KUKA KRL program: Safety_Position.src, Safety_Position.dat

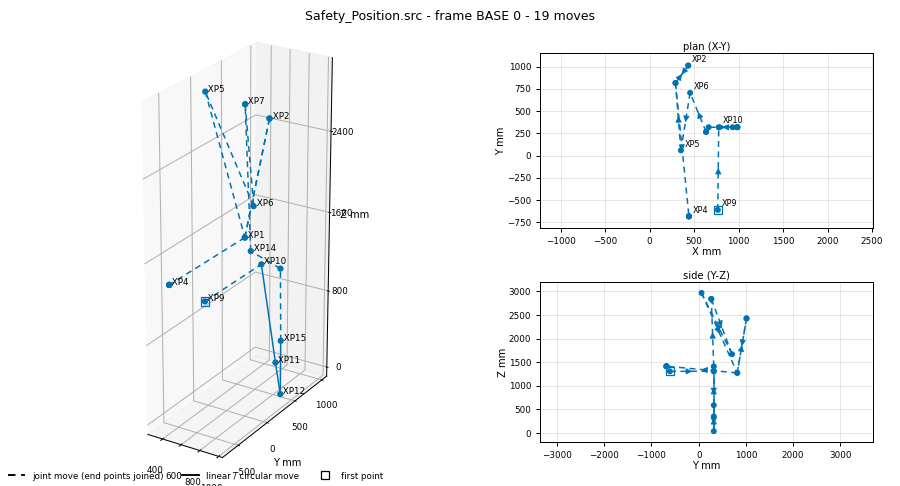
[picture p0: tool path of Safety_Position.src in frame BASE 0, 19 of 19 moves have a stored position in this frame; points joined in program order, loops and branches not executed]
--- Safety_Position.src ---
&ACCESS RVP1
&REL 76
&COMMENT Safety Position
&PARAM DISKPATH = KRC:\R1\Program\Safety Programs
DEF SAFETY_POSITION(DIRECTION :IN,AREA_NR :IN,TYPE_NR :IN )
;FOLD INI
  INT DIRECTION
  INT AREA_NR
  INT TYPE_NR
  decl KrlMsg_T msg
  decl KrlMsgPar_T par[3]
  decl KrlMsgOpt_T opt
  INT nHandle

  IF (DIRECTION>2) OR (DIRECTION<1) THEN
    REPEAT
      msg = {modul[] "Safety Position", nr 1, msg_txt[] "Direction Number Not Valid"}

			opt = {vl_stop true, clear_p_reset true, clear_p_SAW false, log_to_DB false}

			nHandle = Set_KrlMsg(#notify, msg, par[], opt)
      HALT
    UNTIL (DIRECTION<3) AND (DIRECTION>0)
  ENDIF
  IF (AREA_NR>8) OR (AREA_NR<1) THEN
    REPEAT
      msg = {modul[] "Safety Position", nr 2, msg_txt[] "Area Number Not Valid"}

			opt = {vl_stop true, clear_p_reset true, clear_p_SAW false, log_to_DB false}

			nHandle = Set_KrlMsg(#notify, msg, par[], opt)
      HALT
    UNTIL (AREA_NR<9) AND (AREA_NR>0)
  ENDIF
  IF (TYPE_NR>8) OR (TYPE_NR<1) THEN
    REPEAT
  	  msg = {modul[] "Safety Position", nr 1, msg_txt[] "Type Number Not Valid"}

			opt = {vl_stop true, clear_p_reset true, clear_p_SAW false, log_to_DB false}

			nHandle = Set_KrlMsg(#notify, msg, par[], opt)
      HALT
    UNTIL (TYPE_NR<9) AND (TYPE_NR>0)
  ENDIF
  ;ENDFOLD
;===================================================
; MODEL     :CX482
; IE GROUP  :PHEV
; STATION   :110
; ROBOT     :110R1
; FUNCTION  : Safety Position
;================================================

SWITCH AREA_NR

CASE 1  ;AREA 1

  SWITCH TYPE_NR

  CASE 1  ;Area 1 - Safety Position 1
    SWITCH DIRECTION
    CASE 1
    ;Teach here positions from wait area to safety position
    ;check robot movement for collision with other robots
;FOLD PTP P9 CONT Vel=100 % PDAT17 Tool[8]:Gripper_array Base[0];%{PE}%R 8.3.48,%MKUKATPBASIS,%CMOVE,%VPTP,%P 1:PTP, 2:P9, 3:C_DIS, 5:100, 7:PDAT17
$BWDSTART=FALSE
PDAT_ACT=PPDAT17
FDAT_ACT=FP9
BAS(#PTP_PARAMS,100)
PTP XP9 C_DIS
;ENDFOLD
;FOLD PTP P10 CONT Vel=100 % PDAT18 Tool[8]:Gripper_array Base[0];%{PE}%R 8.3.48,%MKUKATPBASIS,%CMOVE,%VPTP,%P 1:PTP, 2:P10, 3:C_DIS, 5:100, 7:PDAT18
$BWDSTART=FALSE
PDAT_ACT=PPDAT18
FDAT_ACT=FP10
BAS(#PTP_PARAMS,100)
PTP XP10 C_DIS
;ENDFOLD
;FOLD LIN P11 CONT Vel=2 m/s CPDAT1 Tool[8]:Gripper_array Base[0];%{PE}%R 8.3.48,%MKUKATPBASIS,%CMOVE,%VLIN,%P 1:LIN, 2:P11, 3:C_DIS C_DIS, 5:2, 7:CPDAT1
$BWDSTART=FALSE
LDAT_ACT=LCPDAT1
FDAT_ACT=FP11
BAS(#CP_PARAMS,2)
LIN XP11 C_DIS C_DIS
;ENDFOLD
;FOLD LIN P12 Vel=2 m/s CPDAT2 Tool[8]:Gripper_array Base[0];%{PE}%R 8.3.48,%MKUKATPBASIS,%CMOVE,%VLIN,%P 1:LIN, 2:P12, 3:, 5:2, 7:CPDAT2
$BWDSTART=FALSE
LDAT_ACT=LCPDAT2
FDAT_ACT=FP12
BAS(#CP_PARAMS,2)
LIN XP12
;ENDFOLD

;abrir gara
cil_bat_reposo()


;FOLD LIN P15 CONT Vel=2 m/s CPDAT3 Tool[8]:Gripper_array Base[0];%{PE}%R 8.3.48,%MKUKATPBASIS,%CMOVE,%VLIN,%P 1:LIN, 2:P15, 3:C_DIS C_DIS, 5:2, 7:CPDAT3
$BWDSTART=FALSE
LDAT_ACT=LCPDAT3
FDAT_ACT=FP15
BAS(#CP_PARAMS,2)
LIN XP15 C_DIS C_DIS
;ENDFOLD
;FOLD PTP P13 CONT Vel=100 % PDAT19 Tool[8]:Gripper_array Base[0];%{PE}%R 8.3.48,%MKUKATPBASIS,%CMOVE,%VPTP,%P 1:PTP, 2:P13, 3:C_DIS, 5:100, 7:PDAT19
$BWDSTART=FALSE
PDAT_ACT=PPDAT19
FDAT_ACT=FP13
BAS(#PTP_PARAMS,100)
PTP XP13 C_DIS
;ENDFOLD
;FOLD PTP P14 CONT Vel=100 % PDAT20 Tool[8]:Gripper_array Base[0];%{PE}%R 8.3.48,%MKUKATPBASIS,%CMOVE,%VPTP,%P 1:PTP, 2:P14, 3:C_DIS, 5:100, 7:PDAT20
$BWDSTART=FALSE
PDAT_ACT=PPDAT20
FDAT_ACT=FP14
BAS(#PTP_PARAMS,100)
PTP XP14 C_DIS
;ENDFOLD

;FOLD PTP P7 Vel=100 % PDAT15 Tool[8]:Gripper_array Base[0];%{PE}%R 8.3.48,%MKUKATPBASIS,%CMOVE,%VPTP,%P 1:PTP, 2:P7, 3:, 5:100, 7:PDAT15
$BWDSTART=FALSE
PDAT_ACT=PPDAT15
FDAT_ACT=FP7
BAS(#PTP_PARAMS,100)
PTP XP7
;ENDFOLD
    CASE 2
    ;Teach here positions from safety position to wait area
;FOLD PTP P8 CONT Vel=100 % PDAT16 Tool[8]:Gripper_array Base[0];%{PE}%R 8.3.48,%MKUKATPBASIS,%CMOVE,%VPTP,%P 1:PTP, 2:P8, 3:C_DIS, 5:100, 7:PDAT16
$BWDSTART=FALSE
PDAT_ACT=PPDAT16
FDAT_ACT=FP8
BAS(#PTP_PARAMS,100)
PTP XP8 C_DIS
;ENDFOLD
    ;check robot movement for collision with other robots
    ENDSWITCH

  CASE 2  ;Area 1 - Safety Position 2

    SWITCH DIRECTION
    CASE 1
;FOLD PTP P6 CONT Vel=100 % PDAT14 Tool[1] Base[0];%{PE}%R 8.3.48,%MKUKATPBASIS,%CMOVE,%VPTP,%P 1:PTP, 2:P6, 3:C_DIS, 5:100, 7:PDAT14
$BWDSTART=FALSE
PDAT_ACT=PPDAT14
FDAT_ACT=FP6
BAS(#PTP_PARAMS,100)
PTP XP6 C_DIS
;ENDFOLD
;FOLD PTP P5 Vel=100 % PDAT13 Tool[1] Base[0];%{PE}%R 8.3.48,%MKUKATPBASIS,%CMOVE,%VPTP,%P 1:PTP, 2:P5, 3:, 5:100, 7:PDAT13
$BWDSTART=FALSE
PDAT_ACT=PPDAT13
FDAT_ACT=FP5
BAS(#PTP_PARAMS,100)
PTP XP5
;ENDFOLD
    ;Teach here positions from waiting area to safety position
    ;check robot movement for collision with other robots
;FOLD PTP P1 Vel=100 % PDAT5 Tool[8]:Gripper_array Base[0];%{PE}%R 8.3.48,%MKUKATPBASIS,%CMOVE,%VPTP,%P 1:PTP, 2:P1, 3:, 5:100, 7:PDAT5
$BWDSTART=FALSE
PDAT_ACT=PPDAT5
FDAT_ACT=FP1
BAS(#PTP_PARAMS,100)
PTP XP1
;ENDFOLD
;FOLD PTP P2 Vel=100 % PDAT6 Tool[8]:Gripper_array Base[0];%{PE}%R 8.3.48,%MKUKATPBASIS,%CMOVE,%VPTP,%P 1:PTP, 2:P2, 3:, 5:100, 7:PDAT6
$BWDSTART=FALSE
PDAT_ACT=PPDAT6
FDAT_ACT=FP2
BAS(#PTP_PARAMS,100)
PTP XP2
;ENDFOLD
    CASE 2
    ;Teach here positions from safety position to waiting area
    ;check robot movement for collision with other robots
;FOLD PTP P2 Vel=100 % PDAT7 Tool[8]:Gripper_array Base[0];%{PE}%R 8.3.48,%MKUKATPBASIS,%CMOVE,%VPTP,%P 1:PTP, 2:P2, 3:, 5:100, 7:PDAT7
$BWDSTART=FALSE
PDAT_ACT=PPDAT7
FDAT_ACT=FP2
BAS(#PTP_PARAMS,100)
PTP XP2
;ENDFOLD
;FOLD PTP P1 Vel=100 % PDAT8 Tool[8]:Gripper_array Base[0];%{PE}%R 8.3.48,%MKUKATPBASIS,%CMOVE,%VPTP,%P 1:PTP, 2:P1, 3:, 5:100, 7:PDAT8
$BWDSTART=FALSE
PDAT_ACT=PPDAT8
FDAT_ACT=FP1
BAS(#PTP_PARAMS,100)
PTP XP1
;ENDFOLD
    ENDSWITCH

  CASE 3  ;Area 1 - Safety Position 3

    SWITCH DIRECTION
    CASE 1
    ;Teach here positions from waiting area to safety position
    ;check robot movement for collision with other robots
;FOLD PTP P4 Vel=100 % PDAT10 Tool[8]:Gripper_array Base[0];%{PE}%R 8.3.48,%MKUKATPBASIS,%CMOVE,%VPTP,%P 1:PTP, 2:P4, 3:, 5:100, 7:PDAT10
$BWDSTART=FALSE
PDAT_ACT=PPDAT10
FDAT_ACT=FP4
BAS(#PTP_PARAMS,100)
PTP XP4
;ENDFOLD
;FOLD PTP P3 Vel=100 % PDAT9 Tool[8]:Gripper_array Base[0];%{PE}%R 8.3.48,%MKUKATPBASIS,%CMOVE,%VPTP,%P 1:PTP, 2:P3, 3:, 5:100, 7:PDAT9
$BWDSTART=FALSE
PDAT_ACT=PPDAT9
FDAT_ACT=FP3
BAS(#PTP_PARAMS,100)
PTP XP3
;ENDFOLD
    CASE 2
    ;Teach here positions from safety position to waiting area
    ;check robot movement for collision with other robots
;FOLD PTP P3 Vel=100 % PDAT11 Tool[8]:Gripper_array Base[0];%{PE}%R 8.3.48,%MKUKATPBASIS,%CMOVE,%VPTP,%P 1:PTP, 2:P3, 3:, 5:100, 7:PDAT11
$BWDSTART=FALSE
PDAT_ACT=PPDAT11
FDAT_ACT=FP3
BAS(#PTP_PARAMS,100)
PTP XP3
;ENDFOLD
;FOLD PTP P4 Vel=100 % PDAT12 Tool[8]:Gripper_array Base[0];%{PE}%R 8.3.48,%MKUKATPBASIS,%CMOVE,%VPTP,%P 1:PTP, 2:P4, 3:, 5:100, 7:PDAT12
$BWDSTART=FALSE
PDAT_ACT=PPDAT12
FDAT_ACT=FP4
BAS(#PTP_PARAMS,100)
PTP XP4
;ENDFOLD
    ENDSWITCH

  CASE 4  ;Area 1 - Safety Position 4

    SWITCH DIRECTION
    CASE 1 ; From Area Request Position To Safety Position
    ;Teach here positions from waiting area to safety position
    ;check robot movement for collision with other robots
    CASE 2 ; From Safety Position To Area Request Position
    ;Teach here positions from safety position to waiting area
    ;check robot movement for collision with other robots
    ENDSWITCH

  CASE 5  ;Area 1 - Safety Position 5

    SWITCH DIRECTION
    CASE 1
    ;Teach here positions from waiting area to safety position
    ;check robot movement for collision with other robots
    CASE 2
    ;Teach here positions from safety position to waiting area
    ;check robot movement for collision with other robots
    ENDSWITCH

  CASE 6  ;Area 1 - Safety Position 6

    SWITCH DIRECTION
    CASE 1
    ;Teach here positions from waiting area to safety position
    ;check robot movement for collision with other robots
    CASE 2
    ;Teach here positions from safety position to waiting area
    ;check robot movement for collision with other robots
    ENDSWITCH

  CASE 7  ;Area 1 - Safety Position 7

    SWITCH DIRECTION
    CASE 1
    ;Teach here positions from waiting area to safety position
    ;check robot movement for collision with other robots
    CASE 2
    ;Teach here positions from safety position to waiting area
    ;check robot movement for collision with other robots
    ENDSWITCH

  CASE 8  ;Area 1 - Safety Position 8

    SWITCH DIRECTION
    CASE 1
    ;Teach here positions from wait area to safety position
    ;check robot movement for collision with other robots
    CASE 2
    ;Teach here positions from safety position to wait area
    ;check robot movement for collision with other robots
    ENDSWITCH

  ENDSWITCH

;====================================================================

CASE 2  ;AREA 2

  SWITCH TYPE_NR
  CASE 1  ;Area 2 - Safety Position 1

    SWITCH DIRECTION
    CASE 1
    ;Teach here pos from waiting area to safety position
    ;check robot movement for collision with other robots
    CASE 2
    ;Teach here positions from safety pos to waiting area
    ;check robot movement for collision with other robots
    ENDSWITCH

  CASE 2  ;Area 2 - Safety Position 2

    SWITCH DIRECTION
    CASE 1
    ;Teach here positions from waiting area to safety position
    ;check robot movement for collision with other robots
    CASE 2
    ;Teach here positions from safety position to waiting area
    ;check robot movement for collision with other robots
    ENDSWITCH

  CASE 3  ;Area 2 - Safety Position 3

    SWITCH DIRECTION
    CASE 1
    ;Teach here positions from waiting area to safety position
    ;check robot movement for collision with other robots
    CASE 2
    ;Teach here positions from safety position to waiting area
    ;check robot movement for collision with other robots
    ENDSWITCH

  CASE 4  ;Area 2 - Safety Position 4

    SWITCH DIRECTION
	  	CASE 1
    ;Teach here positions from waiting area to safety position
    ;check robot movement for collision with other robots
    CASE 2
    ;Teach here positions from safety position to waiting area
    ;check robot movement for collision with other robots
    ENDSWITCH

  CASE 5  ;Area 2 - Safety Position 5

    SWITCH DIRECTION
    CASE 1
    ;Teach here positions from waiting area to safety position
    ;check robot movement for collision with other robots
    CASE 2
    ;Teach here positions from safety position to waiting area
    ;check robot movement for collision with other robots
    ENDSWITCH

  CASE 6    ;Area 2 - Safety Position 6

    SWITCH DIRECTION
    CASE 1
    ;Teach here positions from waiting area to safety position
    ;check robot movement for collision with other robots
    CASE 2
    ;Teach here positions from safety position to waiting area
    ;check robot movement for collision with other robots
    ENDSWITCH

  CASE 7    ;Area 2 - Safety Position 7

    SWITCH DIRECTION
    CASE 1
    ;Teach here positions from waiting area to safety position
    ;check robot movement for collision with other robots
    CASE 2
    ;Teach here positions from safety position to waiting area
    ;check robot movement for collision with other robots
    ENDSWITCH

  CASE 8  ;Area 2 - Safety Position 8

    SWITCH DIRECTION
    CASE 1
    ;Teach here positions from waiting area to safety position
    ;check robot movement for collision with other robots
    CASE 2
    ;Teach here positions from safety position to waiting area
    ;check robot movement for collision with other robots
    ENDSWITCH

  ENDSWITCH

;====================================================================

CASE 3  ;AREA 3

  SWITCH TYPE_NR
  CASE 1  ;Area 3 - Safety Position 1

    SWITCH DIRECTION
    CASE 1
    ;Teach here positions from waiting area to safety position
    ;check robot movement for collision with other robots
    CASE 2
    ;Teach here positions from safety position to waiting area
    ;check robot movement for collision with other robots
    ENDSWITCH

  CASE 2  ;Area 3 - Safety Position 2

    SWITCH DIRECTION
    CASE 1
    ;Teach here positions from waiting area to safety position
    ;check robot movement for collision with other robots
    CASE 2
    ;Teach here positions from safety position to waiting area
    ;check robot movement for collision with other robots
    ENDSWITCH

  CASE 3  ;Area 3 - Safety Position 3

    SWITCH DIRECTION
    CASE 1
    ;Teach here positions from waiting area to safety position
    ;check robot movement for collision with other robots
    CASE 2
    ;Teach here positions from safety position to waiting area
    ;check robot movement for collision with other robots
      ENDSWITCH

  CASE 4  ;Area 3 - Safety Position 4

    SWITCH DIRECTION
    CASE 1
    ;Teach here positions from waiting area to safety position
    ;check robot movement for collision with other robots
    CASE 2
    ;Teach here positions from safety position to waiting area
    ;check robot movement for collision with other robots
    ENDSWITCH

  CASE 5  ;Area 3 - Safety Position 5

    SWITCH DIRECTION
    CASE 1
    ;Teach here positions from waiting area to safety position
    ;check robot movement for collision with other robots
    CASE 2
    ;Teach here positions from safety position to waiting area
    ;check robot movement for collision with other robots
    ENDSWITCH

  CASE 6  ;Area 3 - Safety Position 6

    SWITCH DIRECTION
    CASE 1
    ;Teach here positions from waiting area to safety position
    ;check robot movement for collision with other robots
    CASE 2
    ;Teach here positions from safety position to waiting area
    ;check robot movement for collision with other robots
    ENDSWITCH

  CASE 7  ;Area 3 - Safety Position 7

    SWITCH DIRECTION
    CASE 1
    ;Teach here positions from waiting area to safety position
    ;check robot movement for collision with other robots
    CASE 2
    ;Teach here positions from safety position to waiting area
    ;check robot movement for collision with other robots
    ENDSWITCH

  CASE 8  ;Area 3 - Safety Position 8
    SWITCH DIRECTION
    CASE 1
    ;Teach here positions from waiting area to safety position
    ;check robot movement for collision with other robots
    CASE 2
    ;Teach here positions from safety position to waiting area
    ;check robot movement for collision with other robots
    ENDSWITCH

  ENDSWITCH

;====================================================================

CASE 4  ;AREA 4

  SWITCH TYPE_NR
  CASE 1  ;Area 4 - Safety Position 1

    SWITCH DIRECTION
    CASE 1
		;Teach here positions from waiting area to safety position
		;check robot movement for collision with other robots
		CASE 2
		;Teach here positions from safety position to waiting area
		;check robot movement for collision with other robots

    ENDSWITCH

  CASE 2  ;Area 4 - Safety Position 2

    SWITCH DIRECTION
    CASE 1
	  ;Teach here positions from waiting area to safety position
	  ;check robot movement for collision with other robots
    CASE 2
	  ;Teach here positions from safety position to waiting area
  	;check robot movement for collision with other robots
    ENDSWITCH

  CASE 3  ;Area 4 - Safety Position 3

    SWITCH DIRECTION
    CASE 1
    ;Teach here positions from waiting area to safety position
    ;check robot movement for collision with other robots
    CASE 2
    ;Teach here positions from safety position to waiting area
    ;check robot movement for collision with other robots
    ENDSWITCH

  CASE 4  ;Area 4 - Safety Position 4

    SWITCH DIRECTION
    CASE 1
    ;Teach here positions from waiting area to safety position
    ;check robot movement for collision with other robots
    CASE 2
    ;Teach here positions from safety position to waiting area
    ;check robot movement for collision with other robots
    ENDSWITCH

  CASE 5  ;Area 4 - Safety Position 5

    SWITCH DIRECTION
    CASE 1
    ;Teach here positions from waiting area to safety position
    ;check robot movement for collision with other robots
    CASE 2
    ;Teach here positions from safety position to waiting area
    ;check robot movement for collision with other robots
    ENDSWITCH

  CASE 6  ;Area 4 - Safety Position 6

    SWITCH DIRECTION
    CASE 1
    ;Teach here positions from waiting area to safety position
    ;check robot movement for collision with other robots
    CASE 2
    ;Teach here positions from safety position to waiting area
    ;check robot movement for collision with other robots
    ENDSWITCH

  CASE 7  ;Area 4 - Safety Position 7

    SWITCH DIRECTION
    CASE 1
    ;Teach here positions from waiting area to safety position
    ;check robot movement for collision with other robots
    CASE 2
    ;Teach here positions from safety position to waiting area
    ;check robot movement for collision with other robots
    ENDSWITCH

  CASE 8  ;Area 4 - Safety Position 8

    SWITCH DIRECTION
    CASE 1
    ;Teach here positions from waiting area to safety position
    ;check robot movement for collision with other robots
    CASE 2
    ;Teach here positions from safety position to waiting area
    ;check robot movement for collision with other robots
    ENDSWITCH

  ENDSWITCH

;====================================================================

CASE 5  ;AREA 5

  SWITCH TYPE_NR
  CASE 1  ;Area 5 - Safety Position 1

    SWITCH DIRECTION
    CASE 1
    ;Teach here positions from waiting area to safety position
    ;check robot movement for collision with other robots
    CASE 2
    ;Teach here positions from safety position to waiting area
    ;check robot movement for collision with other robots
    ENDSWITCH

  CASE 2  ;Area 5 - Safety Position 2

    SWITCH DIRECTION
    CASE 1
    ;Teach here positions from waiting area to safety position
    ;check robot movement for collision with other robots
    CASE 2
    ;Teach here positions from safety position to waiting area
    ;check robot movement for collision with other robots
    ENDSWITCH

  CASE 3  ;Area 5 - Safety Position 3

    SWITCH DIRECTION
    CASE 1
    ;Teach here positions from waiting area to safety position
    ;check robot movement for collision with other robots
    CASE 2
    ;Teach here positions from safety position to waiting area
    ;check robot movement for collision with other robots
    ENDSWITCH

  CASE 4  ;Area 5 - Safety Position 4

    SWITCH DIRECTION
    CASE 1
    ;Teach here positions from waiting area to safety position
    ;check robot movement for collision with other robots
    CASE 2
    ;Teach here positions from safety position to waiting area
    ;check robot movement for collision with other robots
    ENDSWITCH

  CASE 5  ;Area 5 - Safety Position 5

    SWITCH DIRECTION
    CASE 1
    ;Teach here positions from waiting area to safety position
    ;check robot movement for collision with other robots
    CASE 2
    ;Teach here positions from safety position to waiting area
    ;check robot movement for collision with other robots
    ENDSWITCH

  CASE 6  ;Area 5 - Safety Position 6

    SWITCH DIRECTION
    CASE 1
    ;Teach here positions from waiting area to safety position
    ;check robot movement for collision with other robots
    CASE 2
    ;Teach here positions from safety position to waiting area
    ;check robot movement for collision with other robots
    ENDSWITCH

  CASE 7  ;Area 5 - Safety Position 7

    SWITCH DIRECTION
    CASE 1
    ;Teach here positions from waiting area to safety position
    ;check robot movement for collision with other robots
    CASE 2
    ;Teach here positions from safety position to waiting area
    ;check robot movement for collision with other robots
    ENDSWITCH

  CASE 8  ;Area 5 - Safety Position 8

    SWITCH DIRECTION
    CASE 1
    ;Teach here positions from waiting area to safety position
    ;check robot movement for collision with other robots
    CASE 2
    ;Teach here positions from safety position to waiting area
    ;check robot movement for collision with other robots
    ENDSWITCH

  ENDSWITCH

;====================================================================

CASE 6  ;AREA 6

  SWITCH TYPE_NR
  CASE 1  ;Area 6 - Safety Position 1

    SWITCH DIRECTION
    CASE 1
    ;Teach here positions from waiting area to safety position
    ;check robot movement for collision with other robots
    CASE 2
    ;Teach here positions from safety position to waiting area
    ;check robot movement for collision with other robots
    ENDSWITCH

  CASE 2  ;Area 6 - Safety Position 2

    SWITCH DIRECTION
    CASE 1
    ;Teach here positions from waiting area to safety position
    ;check robot movement for collision with other robots
    CASE 2
    ;Teach here positions from safety position to waiting area
    ;check robot movement for collision with other robots
    ENDSWITCH

  CASE 3  ;Area 6 - Safety Position 3

    SWITCH DIRECTION
    CASE 1
    ;Teach here positions from waiting area to safety position
    ;check robot movement for collision with other robots
    CASE 2
    ;Teach here positions from safety position to waiting area
    ;check robot movement for collision with other robots
    ENDSWITCH

  CASE 4  ;Area 6 - Safety Position 4

    SWITCH DIRECTION
    CASE 1
    ;Teach here positions from waiting area to safety position
    ;check robot movement for collision with other robots
    CASE 2
    ;Teach here positions from safety position to waiting area
    ;check robot movement for collision with other robots
    ENDSWITCH

  CASE 5  ;Area 6 - Safety Position 5

    SWITCH DIRECTION
    CASE 1
    ;Teach here positions from waiting area to safety position
    ;check robot movement for collision with other robots
    CASE 2
    ;Teach here positions from safety position to waiting area
    ;check robot movement for collision with other robots
    ENDSWITCH

  CASE 6  ;Area 6 - Safety Position 6

    SWITCH DIRECTION
    CASE 1
    ;Teach here positions from waiting area to safety position
    ;check robot movement for collision with other robots
    CASE 2
    ;Teach here positions from safety position to waiting area
    ;check robot movement for collision with other robots
    ENDSWITCH

  CASE 7  ;Area 6 - Safety Position 7

    SWITCH DIRECTION
    CASE 1
    ;Teach here positions from waiting area to safety position
    ;check robot movement for collision with other robots
    CASE 2
    ;Teach here positions from safety position to waiting area
    ;check robot movement for collision with other robots
    ENDSWITCH

  CASE 8  ;Area 6 - Safety Position 8

    SWITCH DIRECTION
    CASE 1
    ;Teach here positions from waiting area to safety position
    ;check robot movement for collision with other robots
    CASE 2
    ;Teach here positions from safety position to waiting area
    ;check robot movement for collision with other robots
    ENDSWITCH

  ENDSWITCH

;====================================================================

CASE 7  ;AREA 7

  SWITCH TYPE_NR
  CASE 1  ;Area 7 - Safety Position 1

    SWITCH DIRECTION
    CASE 1
    ;Teach here positions from waiting area to safety position
    ;check robot movement for collision with other robots
    CASE 2
    ;Teach here positions from safety position to waiting area
    ;check robot movement for collision with other robots
    ENDSWITCH

  CASE 2  ;Area 7 - Safety Position 2

    SWITCH DIRECTION
    CASE 1
    ;Teach here positions from waiting area to safety position
    ;check robot movement for collision with other robots
    CASE 2
    ;Teach here positions from safety position to waiting area
    ;check robot movement for collision with other robots
    ENDSWITCH

  CASE 3  ;Area 7 - Safety Position 3

    SWITCH DIRECTION
    CASE 1
    ;Teach here positions from waiting area to safety position
    ;check robot movement for collision with other robots
    CASE 2
    ;Teach here positions from safety position to waiting area
    ;check robot movement for collision with other robots
    ENDSWITCH

  CASE 4  ;Area 7 - Safety Position 4

    SWITCH DIRECTION
    CASE 1
    ;Teach here positions from waiting area to safety position
    ;check robot movement for collision with other robots
    CASE 2
    ;Teach here positions from safety position to waiting area
    ;check robot movement for collision with other robots
    ENDSWITCH

  CASE 5  ;Area 7 - Safety Position 5

    SWITCH DIRECTION
    CASE 1
    ;Teach here positions from waiting area to safety position
    ;check robot movement for collision with other robots
    CASE 2
    ;Teach here positions from safety position to waiting area
    ;check robot movement for collision with other robots
    ENDSWITCH

  CASE 6  ;Area 7 - Safety Position 6

    SWITCH DIRECTION
    CASE 1
    ;Teach here positions from waiting area to safety position
    ;check robot movement for collision with other robots
    CASE 2
    ;Teach here positions from safety position to waiting area
    ;check robot movement for collision with other robots
    ENDSWITCH

  CASE 7  ;Area 7 - Safety Position 7

    SWITCH DIRECTION
    CASE 1
    ;Teach here positions from waiting area to safety position
    ;check robot movement for collision with other robots
    CASE 2
    ;Teach here positions from safety position to waiting area
    ;check robot movement for collision with other robots
    ENDSWITCH

  CASE 8  ;Area 7 - Safety Position 8

    SWITCH DIRECTION
    CASE 1
    ;Teach here positions from waiting area to safety position
    ;check robot movement for collision with other robots
    CASE 2
    ;Teach here positions from safety position to waiting area
    ;check robot movement for collision with other robots
    ENDSWITCH

  ENDSWITCH

;====================================================================

CASE 8  ;AREA 8

  SWITCH TYPE_NR
  CASE 1  ;Area 8 - Safety Position 1

    SWITCH DIRECTION
    CASE 1
    ;Teach here positions from waiting area to safety position
    ;check robot movement for collision with other robots
    CASE 2
    ;Teach here positions from safety position to waiting area
    ;check robot movement for collision with other robots
    ENDSWITCH

  CASE 2  ;Area 8 - Safety Position 2

    SWITCH DIRECTION
    CASE 1
    ;Teach here positions from waiting area to safety position
    ;check robot movement for collision with other robots
    CASE 2
    ;Teach here positions from safety position to waiting area
    ;check robot movement for collision with other robots
    ENDSWITCH

  CASE 3  ;Area 8 - Safety Position 3

    SWITCH DIRECTION
    CASE 1
    ;Teach here positions from waiting area to safety position
    ;check robot movement for collision with other robots
    CASE 2
    ;Teach here positions from safety position to waiting area
    ;check robot movement for collision with other robots
    ENDSWITCH

  CASE 4  ;Area 8 - Safety Position 4

    SWITCH DIRECTION
    CASE 1
    ;Teach here positions from waiting area to safety position
    ;check robot movement for collision with other robots
    CASE 2
    ;Teach here positions from safety position to waiting area
    ;check robot movement for collision with other robots
    ENDSWITCH

  CASE 5  ;Area 8 - Safety Position 5

    SWITCH DIRECTION
    CASE 1
    ;Teach here positions from waiting area to safety position
    ;check robot movement for collision with other robots
    CASE 2
    ;Teach here positions from safety position to waiting area
    ;check robot movement for collision with other robots
    ENDSWITCH

  CASE 6  ;Area 8 - Safety Position 6

    SWITCH DIRECTION
    CASE 1
    ;Teach here positions from waiting area to safety position
    ;check robot movement for collision with other robots
    CASE 2
    ;Teach here positions from safety position to waiting area
    ;check robot movement for collision with other robots
    ENDSWITCH

  CASE 7  ;Area 8 - Safety Position 7

    SWITCH DIRECTION
    CASE 1
    ;Teach here positions from waiting area to safety position
    ;check robot movement for collision with other robots
    CASE 2
    ;Teach here positions from safety position to waiting area
    ;check robot movement for collision with other robots
    ENDSWITCH

  CASE 8  ;Area 8 - Safety Position 8

    SWITCH DIRECTION
    CASE 1
    ;Teach here positions from waiting area to safety position
    ;check robot movement for collision with other robots
    CASE 2
    ;Teach here positions from safety position to waiting area
    ;check robot movement for collision with other robots
    ENDSWITCH
  ENDSWITCH
ENDSWITCH
END

--- Safety_Position.dat ---
&ACCESS RVP1
&REL 76
&COMMENT Safety Position
&PARAM DISKPATH = KRC:\R1\Program\Safety Programs
DEFDAT  Safety_Position
;FOLD EXTERNAL DECLARATIONS;%{PE}%V3.2.0,%MKUKATPBASIS,%CEXT,%VCOMMON,%P
;FOLD BAS EXT;%{PE}%V3.2.0,%MKUKATPBASIS,%CEXT,%VEXT,%P
EXT  BAS (BAS_COMMAND  :IN,REAL  :IN )
DECL INT SUCCESS
;ENDFOLD
;FOLD GRIPPERTECH EXT
EXT  H50 (INT  :IN,INT  :IN,INT  :IN,GRP_TYP  :IN )
;ENDFOLD (GRIPPERTECH EXT)
;FOLD SPOTTECH EXT
EXT  USERSPOT (S_COMMAND  :IN,SPOT_TYPE  :IN )
;ENDFOLD (SPOTTECH EXT)
;FOLD USER EXT;%{E}%V3.2.0,%MKUKATPUSER,%CEXT,%VEXT,%P
;Make here your modifications
;ENDFOLD
;ENDFOLD

DECL BASIS_SUGG_T LAST_BASIS={POINT1[] "P15                     ",POINT2[] "P15                     ",CP_PARAMS[] "CPDAT3                  ",PTP_PARAMS[] "PDAT20                  ",CONT[] "C_DIS C_DIS             ",CP_VEL[] "2                       ",PTP_VEL[] "100                     ",SYNC_PARAMS[] "SYNCDAT                 ",SPL_NAME[] "S0                      ",A_PARAMS[] "ADAT0                   "}
DECL E6POS XP1={X 290.951233,Y 816.177124,Z 1275.55042,A -86.9976196,B 22.0779018,C -179.006119,S 6,T 27,E1 0.0,E2 0.0,E3 0.0,E4 0.0,E5 0.0,E6 0.0}
DECL FDAT FP1={TOOL_NO 8,BASE_NO 0,IPO_FRAME #BASE,POINT2[] " ",TQ_STATE FALSE}
DECL PDAT PPDAT1={VEL 100.000,ACC 100.000,APO_DIST 100.000,GEAR_JERK 50.0000,EXAX_IGN 0}
DECL E6POS XP2={X 434.240051,Y 1012.69025,Z 2428.93188,A -59.3382492,B 50.5025139,C -135.088516,S 6,T 27,E1 0.0,E2 0.0,E3 0.0,E4 0.0,E5 0.0,E6 0.0}
DECL FDAT FP2={TOOL_NO 8,BASE_NO 0,IPO_FRAME #BASE,POINT2[] " ",TQ_STATE FALSE}
DECL PDAT PPDAT2={VEL 100.000,ACC 100.000,APO_DIST 100.000,GEAR_JERK 50.0000,EXAX_IGN 0}
DECL PDAT PPDAT3={VEL 100.000,ACC 100.000,APO_DIST 100.000,GEAR_JERK 50.0000,EXAX_IGN 0}
DECL PDAT PPDAT4={VEL 100.000,ACC 100.000,APO_DIST 100.000,GEAR_JERK 50.0000,EXAX_IGN 0}
DECL PDAT PPDAT5={VEL 100.000,ACC 100.000,APO_DIST 100.000,GEAR_JERK 50.0000,EXAX_IGN 0}
DECL PDAT PPDAT6={VEL 100.000,ACC 100.000,APO_DIST 100.000,GEAR_JERK 50.0000,EXAX_IGN 0}
DECL PDAT PPDAT7={VEL 100.000,ACC 100.000,APO_DIST 100.000,GEAR_JERK 50.0000,EXAX_IGN 0}
DECL PDAT PPDAT8={VEL 100.000,ACC 100.000,APO_DIST 100.000,GEAR_JERK 50.0000,EXAX_IGN 0}
DECL E6POS XP3={X 442.124359,Y -682.465332,Z 1416.05603,A -171.206314,B 14.8656111,C -154.747955,S 6,T 26,E1 0.0,E2 0.0,E3 0.0,E4 0.0,E5 0.0,E6 0.0}
DECL FDAT FP3={TOOL_NO 8,BASE_NO 0,IPO_FRAME #BASE,POINT2[] " ",TQ_STATE FALSE}
DECL PDAT PPDAT9={VEL 100.000,ACC 100.000,APO_DIST 100.000,GEAR_JERK 50.0000,EXAX_IGN 0}
DECL E6POS XP4={X 442.124359,Y -682.465332,Z 1416.05603,A -171.206314,B 14.8656111,C -154.747955,S 6,T 26,E1 0.0,E2 0.0,E3 0.0,E4 0.0,E5 0.0,E6 0.0}
DECL FDAT FP4={TOOL_NO 8,BASE_NO 0,IPO_FRAME #BASE,POINT2[] " ",TQ_STATE FALSE}
DECL PDAT PPDAT10={VEL 100.000,ACC 100.000,APO_DIST 100.000,GEAR_JERK 50.0000,EXAX_IGN 0}
DECL PDAT PPDAT11={VEL 100.000,ACC 100.000,APO_DIST 100.000,GEAR_JERK 50.0000,EXAX_IGN 0}
DECL PDAT PPDAT12={VEL 100.000,ACC 100.000,APO_DIST 100.000,GEAR_JERK 50.0000,EXAX_IGN 0}
DECL E6POS XP5={X 351.584900,Y 59.7686615,Z 2968.77295,A -75.3211670,B 53.1822166,C -90.1767273,S 6,T 27,E1 0.0,E2 0.0,E3 0.0,E4 0.0,E5 0.0,E6 0.0}
DECL FDAT FP5={TOOL_NO 1,BASE_NO 0,IPO_FRAME #BASE,POINT2[] " ",TQ_STATE FALSE}
DECL PDAT PPDAT13={VEL 100.000,ACC 100.000,APO_DIST 100.000,GEAR_JERK 50.0000,EXAX_IGN 0}
DECL E6POS XP6={X 455.082275,Y 705.701233,Z 1670.91309,A -84.0076447,B 29.3199444,C -172.131531,S 6,T 27,E1 0.0,E2 0.0,E3 0.0,E4 0.0,E5 0.0,E6 0.0}
DECL FDAT FP6={TOOL_NO 1,BASE_NO 0,IPO_FRAME #BASE,POINT2[] " ",TQ_STATE FALSE}
DECL PDAT PPDAT14={VEL 100.000,ACC 100.000,APO_DIST 100.000,APO_MODE #CDIS,GEAR_JERK 50.0000,EXAX_IGN 0}
DECL E6POS XP7={X 634.192505,Y 266.972717,Z 2840.97363,A -75.3211670,B 53.1822166,C -90.1767273,S 6,T 27,E1 0.0,E2 0.0,E3 0.0,E4 0.0,E5 0.0,E6 0.0}
DECL FDAT FP7={TOOL_NO 8,BASE_NO 0,IPO_FRAME #BASE,POINT2[] " ",TQ_STATE FALSE}
DECL PDAT PPDAT15={VEL 100.000,ACC 100.000,APO_DIST 100.000,GEAR_JERK 50.0000,EXAX_IGN 0}
DECL E6POS XP8={X 634.192505,Y 266.972717,Z 2840.97363,A -75.3211670,B 53.1822166,C -90.1767273,S 6,T 27,E1 0.0,E2 0.0,E3 0.0,E4 0.0,E5 0.0,E6 0.0}
DECL FDAT FP8={TOOL_NO 8,BASE_NO 0,IPO_FRAME #BASE,POINT2[] " ",TQ_STATE FALSE}
DECL PDAT PPDAT16={VEL 100.000,ACC 100.000,APO_DIST 100.000,APO_MODE #CDIS,GEAR_JERK 50.0000,EXAX_IGN 0}
DECL E6POS XP9={X 766.503540,Y -609.817139,Z 1308.72668,A 143.540146,B -0.965885580,C -168.571289,S 6,T 26,E1 0.0,E2 0.0,E3 0.0,E4 0.0,E5 0.0,E6 0.0}
DECL FDAT FP9={TOOL_NO 8,BASE_NO 0,IPO_FRAME #BASE,POINT2[] " ",TQ_STATE FALSE}
DECL PDAT PPDAT17={VEL 100.000,ACC 100.000,APO_DIST 100.000,APO_MODE #CDIS,GEAR_JERK 50.0000,EXAX_IGN 0}
DECL E6POS XP10={X 776.451965,Y 319.294281,Z 1308.73560,A -166.737869,B 14.4988384,C -179.106812,S 6,T 27,E1 0.0,E2 0.0,E3 0.0,E4 0.0,E5 0.0,E6 0.0}
DECL FDAT FP10={TOOL_NO 8,BASE_NO 0,IPO_FRAME #BASE,POINT2[] " ",TQ_STATE FALSE}
DECL PDAT PPDAT18={VEL 100.000,ACC 100.000,APO_DIST 100.000,APO_MODE #CDIS,GEAR_JERK 50.0000,EXAX_IGN 0}
DECL E6POS XP11={X 932.907532,Y 319.293732,Z 352.871,A -177.302170,B 0.819990396,C -178.292694,S 6,T 27,E1 0.0,E2 0.0,E3 0.0,E4 0.0,E5 0.0,E6 0.0}
DECL FDAT FP11={TOOL_NO 8,BASE_NO 0,IPO_FRAME #BASE,POINT2[] " ",TQ_STATE FALSE}
DECL LDAT LCPDAT1={VEL 2.00000,ACC 100.000,APO_DIST 100.000,APO_FAC 50.0000,AXIS_VEL 100.000,AXIS_ACC 100.000,ORI_TYP #VAR,CIRC_TYP #BASE,JERK_FAC 50.0000,GEAR_JERK 50.0000,EXAX_IGN 0}
DECL E6POS XP12={X 987.620,Y 319.294037,Z 40.3436966,A -178.391296,B 0.830649495,C -178.657944,S 6,T 27,E1 0.0,E2 0.0,E3 0.0,E4 0.0,E5 0.0,E6 0.0}
DECL FDAT FP12={TOOL_NO 8,BASE_NO 0,IPO_FRAME #BASE,POINT2[] " ",TQ_STATE FALSE}
DECL LDAT LCPDAT2={VEL 2.00000,ACC 100.000,APO_DIST 100.000,APO_FAC 50.0000,AXIS_VEL 100.000,AXIS_ACC 100.000,ORI_TYP #VAR,CIRC_TYP #BASE,JERK_FAC 50.0000,GEAR_JERK 50.0000,EXAX_IGN 0}
DECL E6POS XP13={X 978.002,Y 319.293732,Z 1315.03027,A -177.302170,B 0.819990396,C -178.292694,S 6,T 27,E1 0.0,E2 0.0,E3 0.0,E4 0.0,E5 0.0,E6 0.0}
DECL FDAT FP13={TOOL_NO 8,BASE_NO 0,IPO_FRAME #BASE,POINT2[] " ",TQ_STATE FALSE}
DECL PDAT PPDAT19={VEL 100.000,ACC 100.000,APO_DIST 100.000,APO_MODE #CDIS,GEAR_JERK 50.0000,EXAX_IGN 0}
DECL E6POS XP14={X 663.317871,Y 319.302979,Z 1413.22388,A -177.301712,B 0.699722588,C -178.279175,S 6,T 27,E1 0.0,E2 0.0,E3 0.0,E4 0.0,E5 0.0,E6 0.0}
DECL FDAT FP14={TOOL_NO 8,BASE_NO 0,IPO_FRAME #BASE,POINT2[] " ",TQ_STATE FALSE}
DECL PDAT PPDAT20={VEL 100.000,ACC 100.000,APO_DIST 100.000,APO_MODE #CDIS,GEAR_JERK 50.0000,EXAX_IGN 0}
DECL E6POS XP15={X 987.616577,Y 319.293640,Z 591.502380,A -178.391296,B 0.830655932,C -178.658234,S 6,T 27,E1 0.0,E2 0.0,E3 0.0,E4 0.0,E5 0.0,E6 0.0}
DECL FDAT FP15={TOOL_NO 8,BASE_NO 0,IPO_FRAME #BASE,POINT2[] " ",TQ_STATE FALSE}
DECL LDAT LCPDAT3={VEL 2.00000,ACC 100.000,APO_DIST 100.000,APO_FAC 50.0000,AXIS_VEL 100.000,AXIS_ACC 100.000,ORI_TYP #VAR,CIRC_TYP #BASE,JERK_FAC 50.0000,GEAR_JERK 50.0000,EXAX_IGN 0}
ENDDAT
